PROGRAM Guarding_Safety
VAR
END_VAR

// NETWORK 1

END_PROGRAM

(* stored: Version 1.1.0.1, ProductVersion 3.1.4024.12
   POU Guarding_Safety: Id {b1614d21-cb08-40e0-9274-f1b1d790654c}, SpecialFunc None *)
